VAR_GLOBAL CONSTANT
	valveCount : INT := 10;
	sValveNames : ARRAY[1..valveCount] OF WSTRING := 	["Dilution Selector", 
														"WFI Selector", 
														"Formation Drain", 
														"WFI Filter Bypass Inlet",
														"WFI Filter Inlet",
														"WFI Filter Outlet",
														"WFI Filter Bypass Outlet",
														"Dilution Diverter",
														"Formation Manifold",
														"Suspension Manifold"];	
														
stValveID : ARRAY[1..valveCount] OF INT := 	[1, 	// Dilution Selector
											 2, 		// WFI Selector, 
											 3, 		// Formation Drain, 
											 4, 		// WFI Filter Bypass Inlet,
											 5, 		// WFI Filter Inlet,
											 6, 		// WFI Filter Outlet,
											 7, 		// WFI Filter Bypass Outlet,
											 8, 		// Dilution Diverter,
											 9, 		// Formation Manifold,
											 10 	// Suspension Manifold]
											];	
END_VAR

VAR_GLOBAL

	myText 		: STRING(16) := 'Type';
	myNum		: REAL := 0;
	
	//AO1 AT %Q* : REAL;
	DO1 AT %Q* : BOOL;
	
//---------------------------------- PUMP MAPPING -------------------------------------------------//	
	DO_wfiPump AT %Q* : BOOL;			// Digital Output for turning pump on and off
	AO_wfiPump AT %Q* : REAL;			// Analog Ouput for pump speed control
//-------------------------------------------------------------------------------------------------//

	AI_wfiPressureSensor AT %I* : REAL;			// Analog Ouput for pump speed control


//---------------------------------- CORRIOLIS METER MAPPING -------------------------------------------------//	
	AI_wfiFlowMeter AT %I* : DINT;			// Analog Ouput for pump speed control
//-------------------------------------------------------------------------------------------------//

//---------------------------------- VALVE MAPPING ------------------------------------------------//
	// IOs Dilution Selector Valve (SV)
    DI1_dilutionSV AT %I* : BOOL; 		// Digital Input 1 Closed Feedback
    DI2_dilutionSV AT %I* : BOOL; 		// Digital Input 2 Open Feedback
    AI1_dilutionSV AT %I* : REAL;  		// Analog Input 1 Valve Position Feedback
    DO1_dilutionSV AT %Q* : BOOL; 		// Digital Output 1 Valve Initialization
    AO1_dilutionSV AT %Q* : REAL; 		// Analog Output 1 Valve Position Control Variable (0-10V)
    
    // IOs WFI Selector Valve (SV) 
    DI1_wfiSV AT %I* : BOOL;      		// Digital Input 1 Closed Feedback
    DI2_wfiSV AT %I* : BOOL;      		// Digital Input 2 Open Feedback
    AI1_wfiSV AT %I* : REAL;       		// Analog Input 1 Valve Position Feedback
    DO1_wfiSV AT %Q* : BOOL;     		// Digital Output 1 Valve Initialization
    AO1_wfiSV AT %Q* : REAL;      		// Analog Output 1 Valve Position Control Variable (0-10V)

	// IOs Formation Drain Valve 
    DI1_formDrain AT %I* : BOOL;      	// Digital Input 1 Closed Feedback
    DI2_formDrain AT %I* : BOOL;      	// Digital Input 2 Open Feedback
    AI1_formDrain AT %I* : REAL;       	// Analog Input 1 Valve Position Feedback
    DO1_formDrain AT %Q* : BOOL;     	// Digital Output 1 Valve Initialization
    AO1_formDrain AT %Q* : REAL;      	// Analog Output 1 Valve Position Control Variable (0-10V)
	
	// IOs WFI Bypass Inlet Valve
    DI1_wfiBypassIn AT %I* : BOOL;      // Digital Input 1 Closed Feedback
    DI2_wfiBypassIn AT %I* : BOOL;      // Digital Input 2 Open Feedback
    AI1_wfiBypassIn AT %I* : REAL;      // Analog Input 1 Valve Position Feedback
    DO1_wfiBypassIn AT %Q* : BOOL;     	// Digital Output 1 Valve Initialization
    AO1_wfiBypassIn AT %Q* : REAL;      // Analog Output 1 Valve Position Control Variable (0-10V)
	
		// IOs WFI Filter Inlet Valve
    DI1_wfiFilterIn AT %I* : BOOL;      // Digital Input 1 Closed Feedback
    DI2_wfiFilterIn AT %I* : BOOL;      // Digital Input 2 Open Feedback
    AI1_wfiFilterIn AT %I* : REAL;      // Analog Input 1 Valve Position Feedback
    DO1_wfiFilterIn AT %Q* : BOOL;     	// Digital Output 1 Valve Initialization
    AO1_wfiFilterIn AT %Q* : REAL;      // Analog Output 1 Valve Position Control Variable (0-10V)
	
		// IOs WFI Filter Outlet Valve
    DI1_wfiFilterOut AT %I* : BOOL;      // Digital Input 1 Closed Feedback
    DI2_wfiFilterOut AT %I* : BOOL;      // Digital Input 2 Open Feedback
    AI1_wfiFilterOut AT %I* : REAL;      // Analog Input 1 Valve Position Feedback
    DO1_wfiFilterOut AT %Q* : BOOL;     	// Digital Output 1 Valve Initialization
    AO1_wfiFilterOut AT %Q* : REAL;      // Analog Output 1 Valve Position Control Variable (0-10V)
	
		// IOs WFI Bypass Outlet Valve
    DI1_wfiBypassOut AT %I* : BOOL;      // Digital Input 1 Closed Feedback
    DI2_wfiBypassOut AT %I* : BOOL;      // Digital Input 2 Open Feedback
    AI1_wfiBypassOut AT %I* : REAL;      // Analog Input 1 Valve Position Feedback
    DO1_wfiBypassOut AT %Q* : BOOL;     	// Digital Output 1 Valve Initialization
    AO1_wfiBypassOut AT %Q* : REAL;      // Analog Output 1 Valve Position Control Variable (0-10V)
	
		// IOs Dilution Diverter Valve
    DI1_dilutionDiV AT %I* : BOOL;      // Digital Input 1 Closed Feedback
    DI2_dilutionDiV AT %I* : BOOL;      // Digital Input 2 Open Feedback
    AI1_dilutionDiV AT %I* : REAL;      // Analog Input 1 Valve Position Feedback
    DO1_dilutionDiV AT %Q* : BOOL;     	// Digital Output 1 Valve Initialization
    AO1_dilutionDiV AT %Q* : REAL;      // Analog Output 1 Valve Position Control Variable (0-10V)
	
		// IOs Formation Manifold Valve
    DI1_FormManifold AT %I* : BOOL;      // Digital Input 1 Closed Feedback
    DI2_FormManifold AT %I* : BOOL;      // Digital Input 2 Open Feedback
    AI1_FormManifold AT %I* : REAL;      // Analog Input 1 Valve Position Feedback
    DO1_FormManifold AT %Q* : BOOL;     	// Digital Output 1 Valve Initialization
    AO1_FormManifold AT %Q* : REAL;      // Analog Output 1 Valve Position Control Variable (0-10V)
	
		// IOs Formation Manifold Valve
    DI1_SuspManifold AT %I* : BOOL;      // Digital Input 1 Closed Feedback
    DI2_SuspManifold AT %I* : BOOL;      // Digital Input 2 Open Feedback
    AI1_SuspManifold AT %I* : REAL;      // Analog Input 1 Valve Position Feedback
    DO1_SuspManifold AT %Q* : BOOL;     	// Digital Output 1 Valve Initialization
    AO1_SuspManifold AT %Q* : REAL;      // Analog Output 1 Valve Position Control Variable (0-10V)
//-------------------------------------------------------------------------------------------------//
END_VAR

(* stored: Version 1.1.0.1
   GVL GVL: Id {ae3bfd4d-cad6-090e-2b29-8bdb174a4977} *)
